// This function has been automatically generated from the project information.
{attribute 'signature_flag' := '1073741824'}
{attribute 'TcGenerated'}
{attribute 'no-analysis'}
FUNCTION F_GetTitle : WSTRING
VAR_INPUT
	
END_VAR

F_GetTitle := "TcKNXnetIP_Tunneling_Lib";

END_FUNCTION

(* stored: Version 1.1.0.1
   POU F_GetTitle: Id {d5414a5b-9920-4b59-bd46-91ce0eeeebca}, SpecialFunc None *)
